# EPICS autosave request: motorSimApp/Db/motorSim_positions.req
file "motor_positions.req", P=test:,M=m1
file "motor_positions.req", P=test:,M=m2
file "motor_positions.req", P=test:,M=m3
file "motor_positions.req", P=test:,M=m4
file "motor_positions.req", P=test:,M=m5
file "motor_positions.req", P=test:,M=m6
